PROGRAM POU_1
VAR
END_VAR

//Added Another POu

END_PROGRAM

(* stored: Version 1.1.0.1, ProductVersion 3.1.4024.12
   POU POU_1: Id {13deebe0-5757-48f5-9416-4b29fe9792b1}, SpecialFunc None *)
